PROGRAM PRG_ModbusTest
VAR
	// General	
	bInit					:BOOL := TRUE;
	nForIndex				:INT;
	
	bTestCyclicRead			:BOOL;
	bTestStop				:BOOL;
	bTestReset				:BOOL;
	
	// Modbus
	fbModbus				:FB_ModbusRtuMaster;
	fbModbusBusy			:BOOL;
	fbModbusError			:BOOL;
	
	// Frequency inverters
	aVFD					:ARRAY[1..cNoOfUnits] OF ST_Modbus_Unit; 	
END_VAR
VAR CONSTANT
	cNoOfUnits				:INT:= 2;
	cNoOfParam				:INT:= 4;
END_VAR


// Initialization
//-------------------------------------------	
IF bInit THEN	
	// VFD address 
	aVFD[1].nAddr := 2;
	aVFD[2].nAddr := 3;
	// Parameters to be read in each VFD
	FOR nForIndex := 1 TO cNoOfUnits BY 1 DO
		aVFD[nForIndex].aParam[1].nMemAddr 		:= 1610;	 				 // [W] Power (Value back is in W and not kW)
		aVFD[nForIndex].aParam[1].nQuantity 	:= 4;						 // Bytes
		aVFD[nForIndex].aParam[1].fConvFactor 	:= 10.0; 				     // Conversion index 1 => Conversion factor 10
		aVFD[nForIndex].aParam[1].eDataType 	:= E_Modbus_DataType.eInt32; // Int32
		
		aVFD[nForIndex].aParam[2].nMemAddr 		:= 1612;					// [V] Motor voltage
		aVFD[nForIndex].aParam[2].nQuantity 	:= 2;						// Bytes -> 2 bytes
		aVFD[nForIndex].aParam[2].fConvFactor 	:= 0.1; 					// Conversion index -1 => Conversion factor 0.1
		aVFD[nForIndex].aParam[2].eDataType 	:= E_Modbus_DataType.eInt16;// Int16 
		
		aVFD[nForIndex].aParam[3].nMemAddr 		:= 1613;					// [Hz] Frequency
		aVFD[nForIndex].aParam[3].nQuantity 	:= 2;						// Bytes
		aVFD[nForIndex].aParam[3].fConvFactor 	:= 0.1; 					// Conversion index -1 => Conversion factor 0.1
		aVFD[nForIndex].aParam[3].eDataType 	:= E_Modbus_DataType.eInt16;// Int16 
		
		aVFD[nForIndex].aParam[4].nMemAddr 		:= 1614;					// [A] Motor current 
		aVFD[nForIndex].aParam[4].nQuantity 	:= 4;						// Bytes
		aVFD[nForIndex].aParam[4].fConvFactor 	:= 0.01;				 	// Conversion index -2 => Conversion factor 0.01
		aVFD[nForIndex].aParam[4].eDataType 	:= E_Modbus_DataType.eInt32;// Int32
	END_FOR
	bInit := FALSE;
END_IF


// Update function block that handles modbus communication
//-------------------------------------------	
fbModbus(
	pUnit:= ADR(aVFD),
	nNoOfUnits := cNoOfUnits,
	nNoOfParam := cNoOfParam,
	bBusy => fbModbusBusy,
	bError => fbModbusError);

	
// Commands	
//-------------------------------------------		
// Test/Start cyclic read of data
IF bTestCyclicRead THEN
	fbModbus.M_CmdCyclicRead();
	bTestCyclicRead := FALSE;
END_IF

// Stop cyclic read of data
IF bTestStop THEN
	fbModbus.M_CmdStop();
	bTestStop := FALSE;
END_IF

// Reset of error
IF bTestReset THEN
	fbModbus.M_CmdReset();
	bTestReset := FALSE;
END_IF

	
// Results (Read outs)
//-------------------------------------
// VFD 1
//aVFD[1].aParam[1].aDataValue;		// [W] Power
//aVFD[1].aParam[2].aDataValue;		// [V] Motor voltage
//aVFD[1].aParam[3].aDataValue;		// [Hz] Frequency
//aVFD[1].aParam[4].aDataValue;		// [A] Motor current 

// VFD 2
//aVFD[2].aParam[1].aDataValue;		// [W] Power
//aVFD[2].aParam[2].aDataValue;		// [V] Motor voltage
//aVFD[2].aParam[3].aDataValue;		// [Hz] Frequency
//aVFD[2].aParam[4].aDataValue;		// [A] Motor current

END_PROGRAM

(* stored: Version 1.1.0.1, ProductVersion 3.1.4024.12
   POU PRG_ModbusTest: Id {e325ca49-fd54-4936-bce4-96a1102c65e7}, SpecialFunc None *)
